KUKA KRL program: MODULO.src

&ACCESS RV
&PARAM TEMPLATE = C:\KRC\Roboter\Template\FunctionVorgabe
&PARAM EDITMASK = *
DEFFCT INT modulo(n :IN, m :IN)
DECL INT n, m

  IF (n == 0) OR (m == 0) THEN
    RETURN 0
  ENDIF
  RETURN n - ( n / m ) * m

ENDFCT
